// TIA Portal V16 export
// export: Created 2021-06-17T11:14:34.1766954Z, ExportSetting WithDefaults, DisplayName Totally Integrated Automation Portal, DisplayVersion V16 Update 4, DisplayName TIA Portal Version Control Interface, DisplayVersion V16 Update 2, DisplayName TIA Portal Openness, DisplayVersion V16 Update 4, DisplayName SINAMICS Startdrive Advanced, DisplayVersion V16 Update 5, DisplayName SINAMICS Startdrive G130, G150, S120, S150, SINAMICS MV, S210, DisplayVersion V16 Update 5, DisplayName SINAMICS Startdrive G110M, G120, G120C, G120D, G120P, G115D, DisplayVersion V16 Update 5, DisplayName STEP 7 Professional, DisplayVersion V16 Update 4, DisplayName SIMATIC Energy Suite, DisplayVersion V16 Update 4, DisplayName STEP 7 Safety, DisplayVersion V16, DisplayName WinCC Advanced / Unified PC, DisplayVersion V16 Update 4, DisplayName SIMATIC Visualization Architect, DisplayVersion V16 Update 1
TYPE "udt_EM480V_DS_142"
// RDREC
// ● Data record DS 142 for basic measured values (read only).
// stored: IsFailsafeCompliant false
   STRUCT
      "version" { ExternalWritable := 'False'} : Byte;
      reserved { ExternalWritable := 'False'} : Byte;
      uL1N { ExternalWritable := 'False'} : Real;   // Voltage UL1-N, V
      uL2N { ExternalWritable := 'False'} : Real;   // Voltage UL2-N, V
      uL3N { ExternalWritable := 'False'} : Real;   // Voltage UL3-N, V
      uL12 { ExternalWritable := 'False'} : Real;   // Voltage UL1-L2, V
      uL23 { ExternalWritable := 'False'} : Real;   // Voltage UL2-L3, V
      uL31 { ExternalWritable := 'False'} : Real;   // Voltage UL3-L1, V
      iL1 { ExternalWritable := 'False'} : Real;   // Current L1, A
      iL2 { ExternalWritable := 'False'} : Real;   // Current L2, A
      iL3 { ExternalWritable := 'False'} : Real;   // Current L3, A
      pfL1 { ExternalWritable := 'False'} : Real;   // Power factor L1
      pfL2 { ExternalWritable := 'False'} : Real;   // Power factor L2
      pfL3 { ExternalWritable := 'False'} : Real;   // Power factor L3
      pfTotal { ExternalWritable := 'False'} : Real;   // Total power factor L1L2L3
      frequency { ExternalWritable := 'False'} : Real;   // Frequency, Hz
      amplitudeUnbalanceForVoltage { ExternalWritable := 'False'} : Real;   // Amplitude unbalance for voltage, %
      amplitudeUnbalanceForCurrent { ExternalWritable := 'False'} : Real;   // Amplitude unbalance for current, %
      sL1 { ExternalWritable := 'False'} : Real;   // Apparent power L1, VA
      sL2 { ExternalWritable := 'False'} : Real;   // Apparent power L2, VA
      sL3 { ExternalWritable := 'False'} : Real;   // Apparent power L3, VA
      sTotal { ExternalWritable := 'False'} : Real;   // Total apparent power L1L2L3, VA
      qL1 { ExternalWritable := 'False'} : Real;   // Reactive power L1, var
      qL2 { ExternalWritable := 'False'} : Real;   // Reactive power L2, var
      qL3 { ExternalWritable := 'False'} : Real;   // Reactive power L3, var
      qTotal { ExternalWritable := 'False'} : Real;   // Total reactive power L1L2L3, var
      pL1 { ExternalWritable := 'False'} : Real;   // Active power L1, W
      pL2 { ExternalWritable := 'False'} : Real;   // Active power L2, W
      pL3 { ExternalWritable := 'False'} : Real;   // Active power L3, W
      pTotal { ExternalWritable := 'False'} : Real;   // Total active power L1L2L3, W
      phaseAngleL1 { ExternalWritable := 'False'} : Real;   // Phase angle L1, °
      phaseAngleL2 { ExternalWritable := 'False'} : Real;   // Phase angle L2, °
      phaseAngleL3 { ExternalWritable := 'False'} : Real;   // Phase angle L3, °
      appEnTotal { ExternalWritable := 'False'} : Real;   // Total apparent energy L1L2L3, VAh
      reactEnTotal { ExternalWritable := 'False'} : Real;   // Total reactive energy L1L2L3, VAh
      actEnTotal { ExternalWritable := 'False'} : Real;   // Total active energy L1L2L3, Wh
      reactEnInflow { ExternalWritable := 'False'} : Real;   // Total reactive energy inflow L1L2L3, varh
      reactEnOutflow { ExternalWritable := 'False'} : Real;   // Total reactive energy outflow L1L2L3, varh
      actEnInflow { ExternalWritable := 'False'} : Real;   // Total active energy inflow L1L2L3, Wh
      actEnOutflow { ExternalWritable := 'False'} : Real;   // Total active energy outflow L1L2L3, Wh
      appEnTotalLR { ExternalWritable := 'False'} : LReal;   // Total apparent energy L1L2L3, VAh
      reactEnTotalLR { ExternalWritable := 'False'} : LReal;   // Total reactive energy L1L2L3, varh
      actEnTotalLR { ExternalWritable := 'False'} : LReal;   // Total active energy L1L2L3, Wh
      reactEnInflowLR { ExternalWritable := 'False'} : LReal;   // Total reactive energy inflow L1L2L3, varh
      reactEnOutflowLR { ExternalWritable := 'False'} : LReal;   // Total reactive energy outflow L1L2L3, varh
      actEnInflowLR { ExternalWritable := 'False'} : LReal;   // Total active energy inflow L1L2L3, Wh
      actEnOutflowLR { ExternalWritable := 'False'} : LReal;   // Total active energy outflow L1L2L3, Wh
      iNeutral { ExternalWritable := 'False'} : Real;   // Neutral current, A
   END_STRUCT;
END_TYPE
